% RSLogix 500 project 003.RSS, saved by version 8.30.00.16 %
PROJECT "UNTITLED"    % processor: Bul.1763 MicroLogix 1100 Series B %

PROGRAM FILES
  LAD 2 "MAIN"  2 rungs
  LAD 3 "ALARMS"  1 rungs
  LAD 4 "IO"  4 rungs

DATA FILES
  O0 OUTPUT  5 elements
  I1 INPUT  7 elements
  S2 STATUS  66 elements
  B3 BINARY  1 elements
  T4 TIMER  1 elements
  C5 COUNTER  1 elements
  R6 CONTROL  1 elements
  N7 INTEGER  1 elements
  F8 FLOAT  1 elements

LADDER 2 "MAIN"
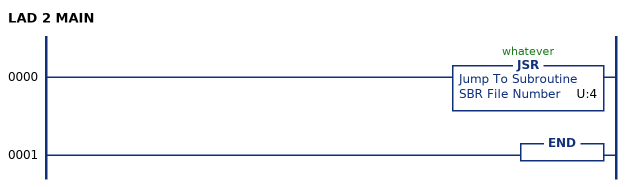
% Rung: 0 %
SOR JSR U:4 EOR
%   U:4  "whatever" %
% Rung: 1 %
SOR END EOR

LADDER 4 "IO"
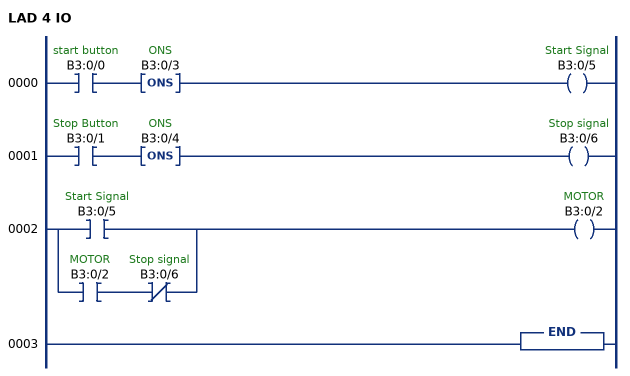
% Rung: 0 %
SOR XIC B3:0/0 ONS B3:0/3 OTE B3:0/5 EOR
%   B3:0/0  "start button" %
%   B3:0/3  "ONS" %
%   B3:0/5  "Start Signal" %
% Rung: 1 %
SOR XIC B3:0/1 ONS B3:0/4 OTE B3:0/6 EOR
%   B3:0/1  "Stop Button" %
%   B3:0/4  "ONS" %
%   B3:0/6  "Stop signal" %
% Rung: 2 %
SOR BST XIC B3:0/5 NXB XIC B3:0/2 XIO B3:0/6 BND OTE B3:0/2 EOR
%   B3:0/5  "Start Signal" %
%   B3:0/2  "MOTOR" %
%   B3:0/6  "Stop signal" %
% Rung: 3 %
SOR END EOR

REVISION NOTES
  0: motor test
